FUNCTION_BLOCK FB_Complex
VAR
	_fMember 		: LREAL := 67.5;
	_stMember 		: ST_Complex := (bMember := TRUE, eMember := E_Enum.Member2, arrfMember := [1.23, 3.33, 1.11]); 
	_fbSimpleMember : FB_Simple(TRUE, 78, 'Complex Test.');
	_fbPackedMember : FB_Packed;
END_VAR

END_FUNCTION_BLOCK

(* stored: Version 1.1.0.1
   POU FB_Complex: Id {e45034a7-979a-4ae9-ad47-43216a229aae}, SpecialFunc None *)
